{attribute 'pack_mode' := '1'}
TYPE ST_ClearAllFaults EXTENDS ST_MsgToPLC:
STRUCT
END_STRUCT
END_TYPE

(* stored: Version 1.1.0.1, ProductVersion 3.1.4022.18
   DUT ST_ClearAllFaults: Id {22b33a8d-6641-48b7-9d12-c323dd2cf817} *)
